VAR_GLOBAL CONSTANT
    PI : LREAL := 3.14159265358979;
END_VAR

(* stored: Version 1.1.0.1
   GVL GVL_Constants: Id {3ba0174e-b0db-43a1-86d2-d8814f3d1e3c} *)
